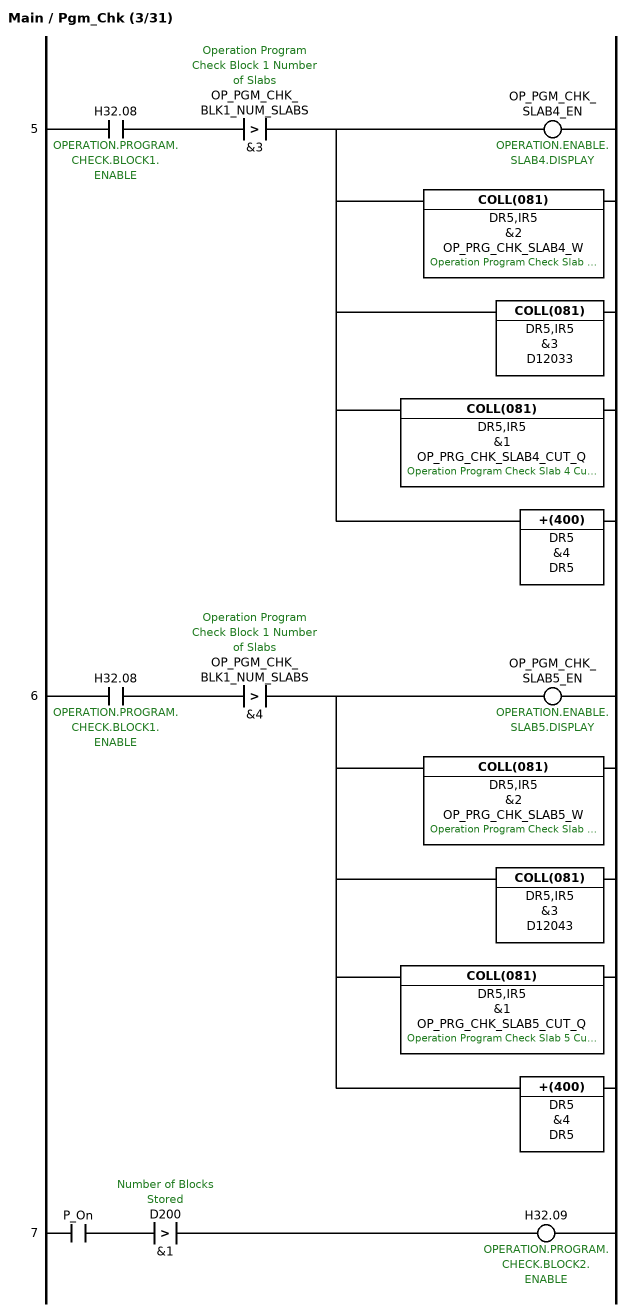
; [picture p96: Main / Pgm_Chk, rungs 5-7]
; rung 5
LD H32.08  ; OPERATION.PROGRAM.CHECK.BLOCK1.ENABLE
AND>(320) OP_PGM_CHK_BLK1_NUM_SLABS &3  ; Operation Program Check Block 1 Number of Slabs
OUT OP_PGM_CHK_SLAB4_EN  ; OPERATION.ENABLE.SLAB4.DISPLAY
COLL(081) DR5,IR5 &2 OP_PRG_CHK_SLAB4_W  ; Operation Program Check Slab 4 Width
COLL(081) DR5,IR5 &3 D12033
COLL(081) DR5,IR5 &1 OP_PRG_CHK_SLAB4_CUT_Q  ; Operation Program Check Slab 4 Cut Quantity
+(400) DR5 &4 DR5
; rung 6
LD H32.08  ; OPERATION.PROGRAM.CHECK.BLOCK1.ENABLE
AND>(320) OP_PGM_CHK_BLK1_NUM_SLABS &4  ; Operation Program Check Block 1 Number of Slabs
OUT OP_PGM_CHK_SLAB5_EN  ; OPERATION.ENABLE.SLAB5.DISPLAY
COLL(081) DR5,IR5 &2 OP_PRG_CHK_SLAB5_W  ; Operation Program Check Slab 5 Width
COLL(081) DR5,IR5 &3 D12043
COLL(081) DR5,IR5 &1 OP_PRG_CHK_SLAB5_CUT_Q  ; Operation Program Check Slab 5 Cut Quantity
+(400) DR5 &4 DR5
; rung 7
LD P_On
AND>(320) D200 &1  ; Number of Blocks Stored
OUT H32.09  ; OPERATION.PROGRAM.CHECK.BLOCK2.ENABLE

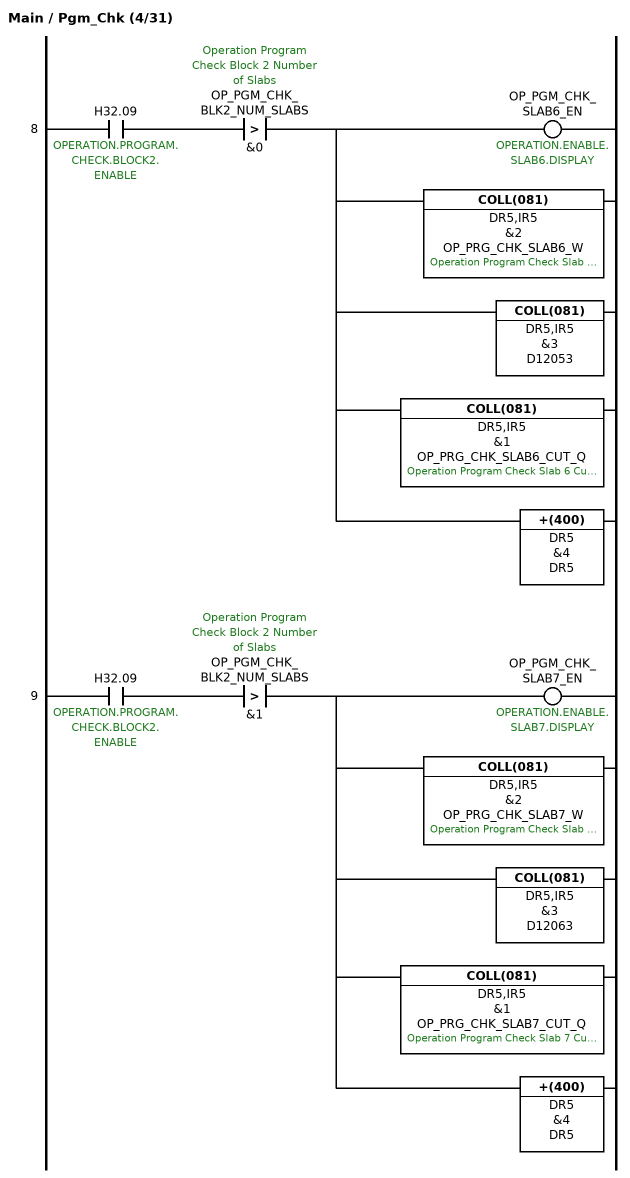
; rung 8
LD H32.09  ; OPERATION.PROGRAM.CHECK.BLOCK2.ENABLE
AND>(320) OP_PGM_CHK_BLK2_NUM_SLABS &0  ; Operation Program Check Block 2 Number of Slabs
OUT OP_PGM_CHK_SLAB6_EN  ; OPERATION.ENABLE.SLAB6.DISPLAY
COLL(081) DR5,IR5 &2 OP_PRG_CHK_SLAB6_W  ; Operation Program Check Slab 6 Width
COLL(081) DR5,IR5 &3 D12053
COLL(081) DR5,IR5 &1 OP_PRG_CHK_SLAB6_CUT_Q  ; Operation Program Check Slab 6 Cut Quantity
+(400) DR5 &4 DR5
; rung 9
LD H32.09  ; OPERATION.PROGRAM.CHECK.BLOCK2.ENABLE
AND>(320) OP_PGM_CHK_BLK2_NUM_SLABS &1  ; Operation Program Check Block 2 Number of Slabs
OUT OP_PGM_CHK_SLAB7_EN  ; OPERATION.ENABLE.SLAB7.DISPLAY
COLL(081) DR5,IR5 &2 OP_PRG_CHK_SLAB7_W  ; Operation Program Check Slab 7 Width
COLL(081) DR5,IR5 &3 D12063
COLL(081) DR5,IR5 &1 OP_PRG_CHK_SLAB7_CUT_Q  ; Operation Program Check Slab 7 Cut Quantity
+(400) DR5 &4 DR5

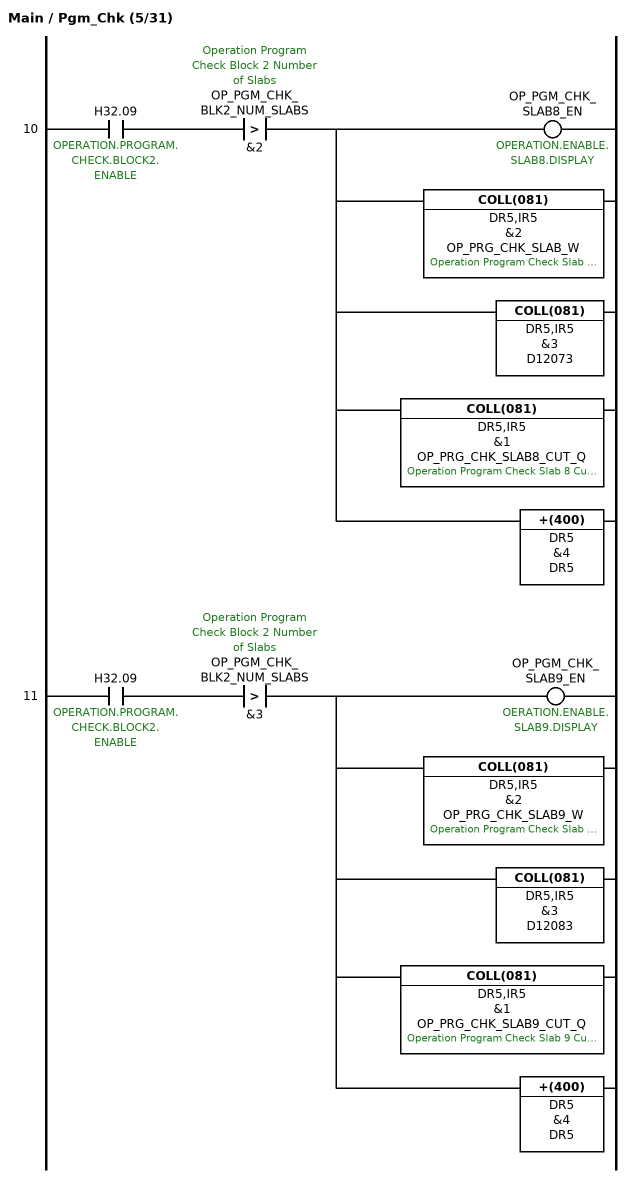
; rung 10
LD H32.09  ; OPERATION.PROGRAM.CHECK.BLOCK2.ENABLE
AND>(320) OP_PGM_CHK_BLK2_NUM_SLABS &2  ; Operation Program Check Block 2 Number of Slabs
OUT OP_PGM_CHK_SLAB8_EN  ; OPERATION.ENABLE.SLAB8.DISPLAY
COLL(081) DR5,IR5 &2 OP_PRG_CHK_SLAB_W  ; Operation Program Check Slab 8 Width
COLL(081) DR5,IR5 &3 D12073
COLL(081) DR5,IR5 &1 OP_PRG_CHK_SLAB8_CUT_Q  ; Operation Program Check Slab 8 Cut Quantity
+(400) DR5 &4 DR5
; rung 11
LD H32.09  ; OPERATION.PROGRAM.CHECK.BLOCK2.ENABLE
AND>(320) OP_PGM_CHK_BLK2_NUM_SLABS &3  ; Operation Program Check Block 2 Number of Slabs
OUT OP_PGM_CHK_SLAB9_EN  ; OERATION.ENABLE.SLAB9.DISPLAY
COLL(081) DR5,IR5 &2 OP_PRG_CHK_SLAB9_W  ; Operation Program Check Slab 9 Width
COLL(081) DR5,IR5 &3 D12083
COLL(081) DR5,IR5 &1 OP_PRG_CHK_SLAB9_CUT_Q  ; Operation Program Check Slab 9 Cut Quantity
+(400) DR5 &4 DR5

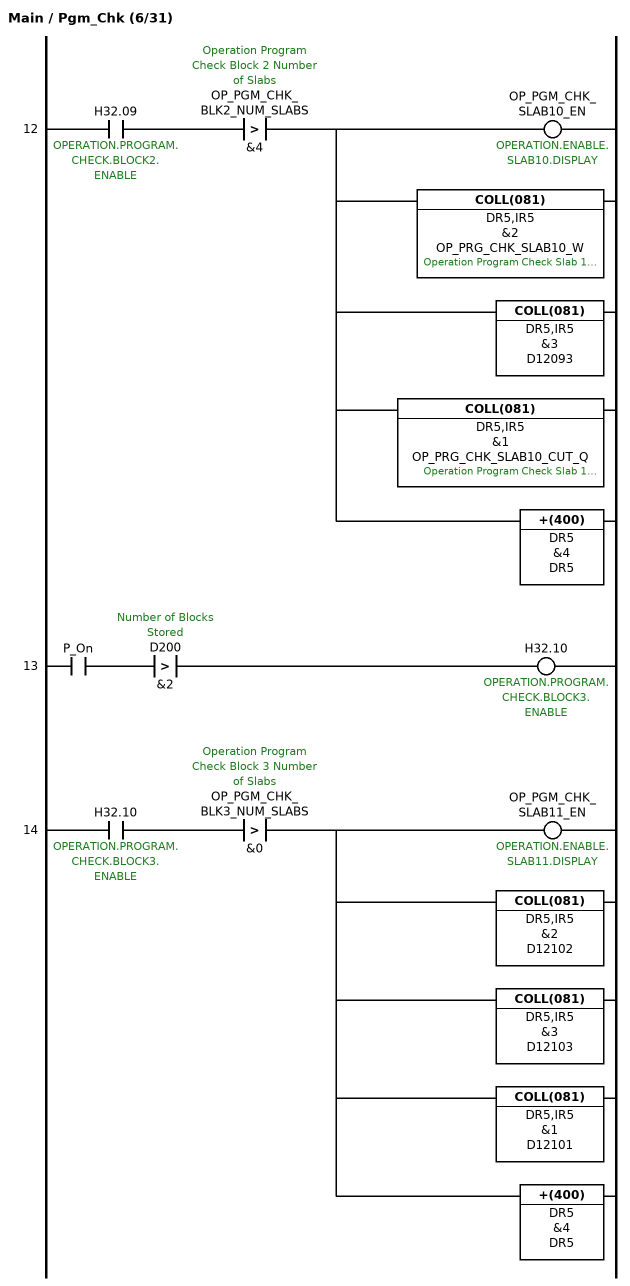
; rung 12
LD H32.09  ; OPERATION.PROGRAM.CHECK.BLOCK2.ENABLE
AND>(320) OP_PGM_CHK_BLK2_NUM_SLABS &4  ; Operation Program Check Block 2 Number of Slabs
OUT OP_PGM_CHK_SLAB10_EN  ; OPERATION.ENABLE.SLAB10.DISPLAY
COLL(081) DR5,IR5 &2 OP_PRG_CHK_SLAB10_W  ; Operation Program Check Slab 10 Width
COLL(081) DR5,IR5 &3 D12093
COLL(081) DR5,IR5 &1 OP_PRG_CHK_SLAB10_CUT_Q  ; Operation Program Check Slab 10 Cut Quantity
+(400) DR5 &4 DR5
; rung 13
LD P_On
AND>(320) D200 &2  ; Number of Blocks Stored
OUT H32.10  ; OPERATION.PROGRAM.CHECK.BLOCK3.ENABLE
; rung 14
LD H32.10  ; OPERATION.PROGRAM.CHECK.BLOCK3.ENABLE
AND>(320) OP_PGM_CHK_BLK3_NUM_SLABS &0  ; Operation Program Check Block 3 Number of Slabs
OUT OP_PGM_CHK_SLAB11_EN  ; OPERATION.ENABLE.SLAB11.DISPLAY
COLL(081) DR5,IR5 &2 D12102
COLL(081) DR5,IR5 &3 D12103
COLL(081) DR5,IR5 &1 D12101
+(400) DR5 &4 DR5

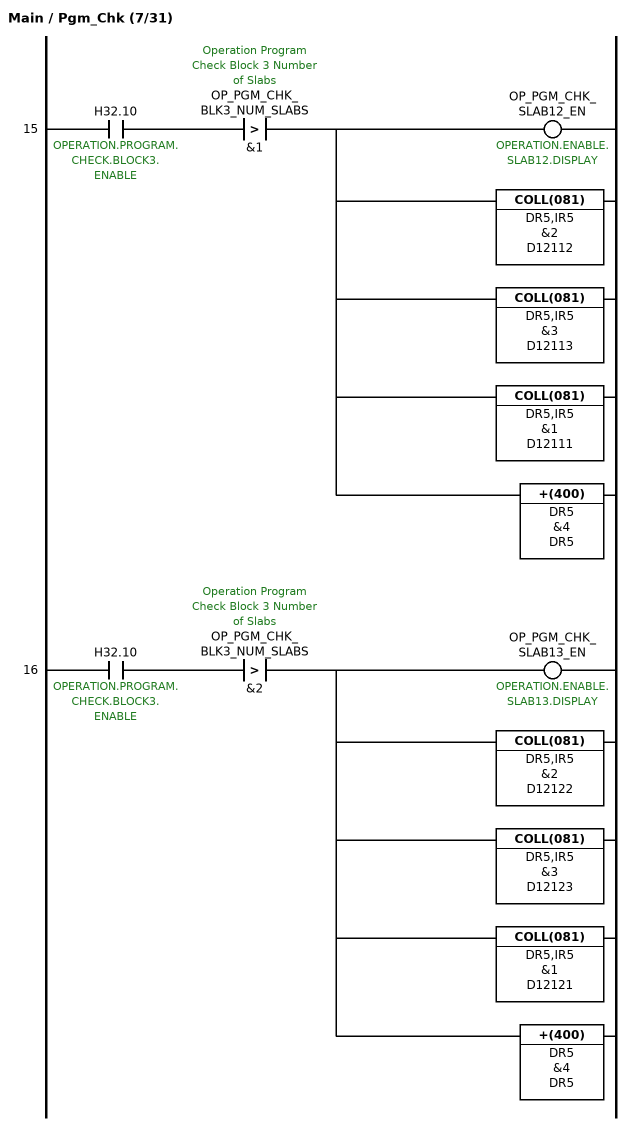
; rung 15
LD H32.10  ; OPERATION.PROGRAM.CHECK.BLOCK3.ENABLE
AND>(320) OP_PGM_CHK_BLK3_NUM_SLABS &1  ; Operation Program Check Block 3 Number of Slabs
OUT OP_PGM_CHK_SLAB12_EN  ; OPERATION.ENABLE.SLAB12.DISPLAY
COLL(081) DR5,IR5 &2 D12112
COLL(081) DR5,IR5 &3 D12113
COLL(081) DR5,IR5 &1 D12111
+(400) DR5 &4 DR5
; rung 16
LD H32.10  ; OPERATION.PROGRAM.CHECK.BLOCK3.ENABLE
AND>(320) OP_PGM_CHK_BLK3_NUM_SLABS &2  ; Operation Program Check Block 3 Number of Slabs
OUT OP_PGM_CHK_SLAB13_EN  ; OPERATION.ENABLE.SLAB13.DISPLAY
COLL(081) DR5,IR5 &2 D12122
COLL(081) DR5,IR5 &3 D12123
COLL(081) DR5,IR5 &1 D12121
+(400) DR5 &4 DR5

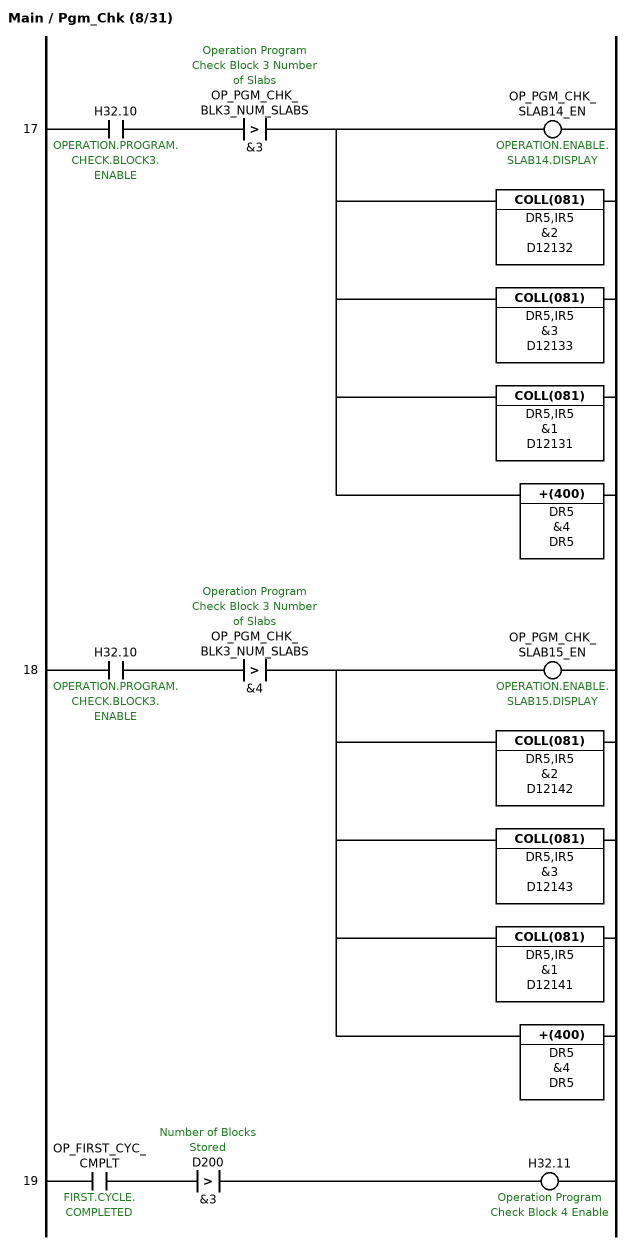
; rung 17
LD H32.10  ; OPERATION.PROGRAM.CHECK.BLOCK3.ENABLE
AND>(320) OP_PGM_CHK_BLK3_NUM_SLABS &3  ; Operation Program Check Block 3 Number of Slabs
OUT OP_PGM_CHK_SLAB14_EN  ; OPERATION.ENABLE.SLAB14.DISPLAY
COLL(081) DR5,IR5 &2 D12132
COLL(081) DR5,IR5 &3 D12133
COLL(081) DR5,IR5 &1 D12131
+(400) DR5 &4 DR5
; rung 18
LD H32.10  ; OPERATION.PROGRAM.CHECK.BLOCK3.ENABLE
AND>(320) OP_PGM_CHK_BLK3_NUM_SLABS &4  ; Operation Program Check Block 3 Number of Slabs
OUT OP_PGM_CHK_SLAB15_EN  ; OPERATION.ENABLE.SLAB15.DISPLAY
COLL(081) DR5,IR5 &2 D12142
COLL(081) DR5,IR5 &3 D12143
COLL(081) DR5,IR5 &1 D12141
+(400) DR5 &4 DR5
; rung 19
LD OP_FIRST_CYC_CMPLT  ; FIRST.CYCLE.COMPLETED
AND>(320) D200 &3  ; Number of Blocks Stored
OUT H32.11  ; Operation Program Check Block 4 Enable

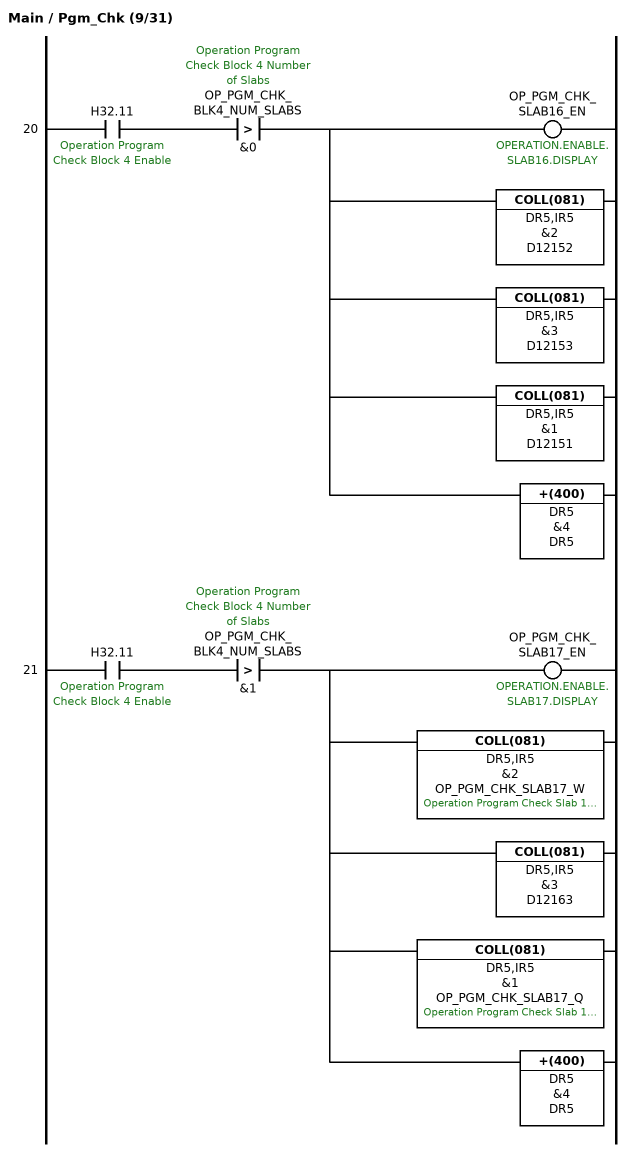
; rung 20
LD H32.11  ; Operation Program Check Block 4 Enable
AND>(320) OP_PGM_CHK_BLK4_NUM_SLABS &0  ; Operation Program Check Block 4 Number of Slabs
OUT OP_PGM_CHK_SLAB16_EN  ; OPERATION.ENABLE.SLAB16.DISPLAY
COLL(081) DR5,IR5 &2 D12152
COLL(081) DR5,IR5 &3 D12153
COLL(081) DR5,IR5 &1 D12151
+(400) DR5 &4 DR5
; rung 21
LD H32.11  ; Operation Program Check Block 4 Enable
AND>(320) OP_PGM_CHK_BLK4_NUM_SLABS &1  ; Operation Program Check Block 4 Number of Slabs
OUT OP_PGM_CHK_SLAB17_EN  ; OPERATION.ENABLE.SLAB17.DISPLAY
COLL(081) DR5,IR5 &2 OP_PGM_CHK_SLAB17_W  ; Operation Program Check Slab 17 Size
COLL(081) DR5,IR5 &3 D12163
COLL(081) DR5,IR5 &1 OP_PGM_CHK_SLAB17_Q  ; Operation Program Check Slab 17 Quantity
+(400) DR5 &4 DR5

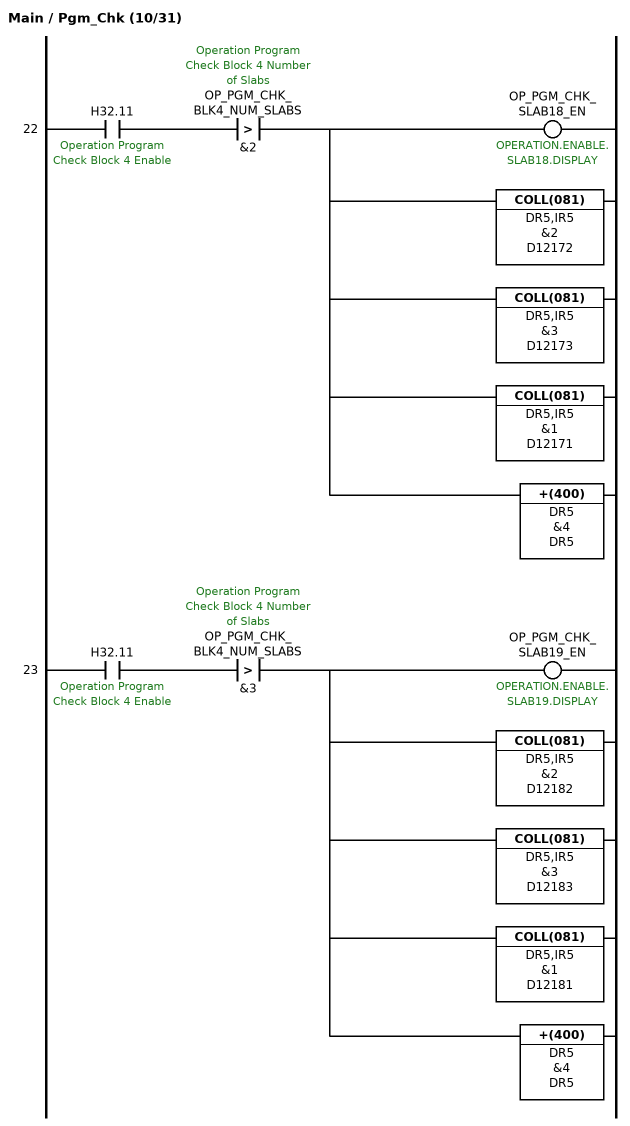
; rung 22
LD H32.11  ; Operation Program Check Block 4 Enable
AND>(320) OP_PGM_CHK_BLK4_NUM_SLABS &2  ; Operation Program Check Block 4 Number of Slabs
OUT OP_PGM_CHK_SLAB18_EN  ; OPERATION.ENABLE.SLAB18.DISPLAY
COLL(081) DR5,IR5 &2 D12172
COLL(081) DR5,IR5 &3 D12173
COLL(081) DR5,IR5 &1 D12171
+(400) DR5 &4 DR5
; rung 23
LD H32.11  ; Operation Program Check Block 4 Enable
AND>(320) OP_PGM_CHK_BLK4_NUM_SLABS &3  ; Operation Program Check Block 4 Number of Slabs
OUT OP_PGM_CHK_SLAB19_EN  ; OPERATION.ENABLE.SLAB19.DISPLAY
COLL(081) DR5,IR5 &2 D12182
COLL(081) DR5,IR5 &3 D12183
COLL(081) DR5,IR5 &1 D12181
+(400) DR5 &4 DR5

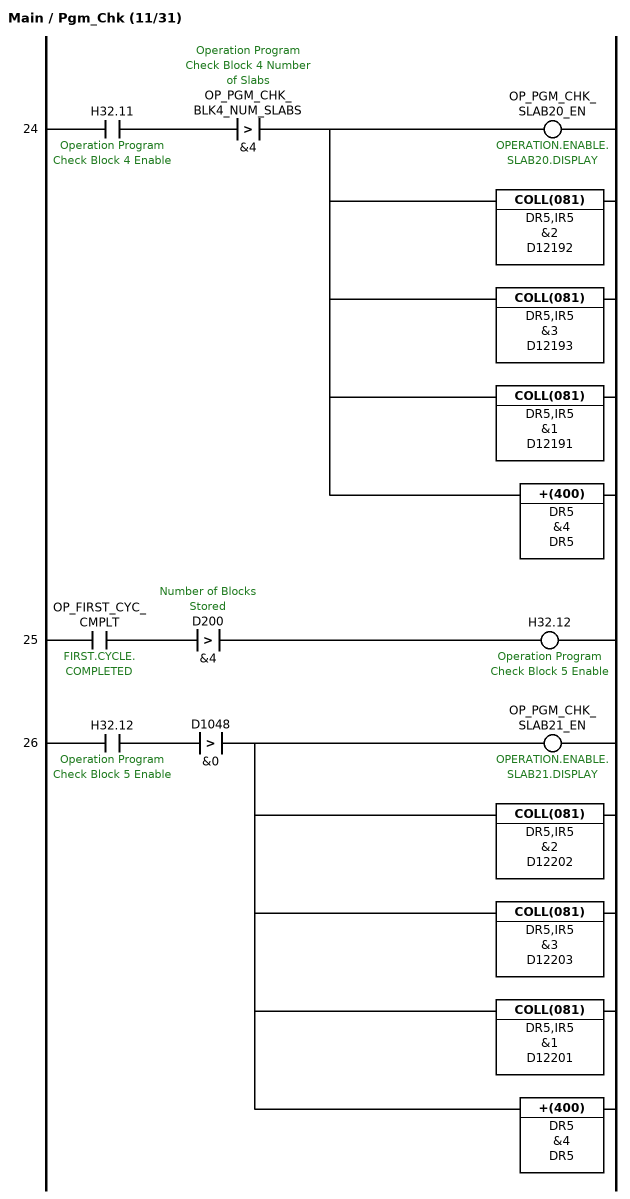
; rung 24
LD H32.11  ; Operation Program Check Block 4 Enable
AND>(320) OP_PGM_CHK_BLK4_NUM_SLABS &4  ; Operation Program Check Block 4 Number of Slabs
OUT OP_PGM_CHK_SLAB20_EN  ; OPERATION.ENABLE.SLAB20.DISPLAY
COLL(081) DR5,IR5 &2 D12192
COLL(081) DR5,IR5 &3 D12193
COLL(081) DR5,IR5 &1 D12191
+(400) DR5 &4 DR5
; rung 25
LD OP_FIRST_CYC_CMPLT  ; FIRST.CYCLE.COMPLETED
AND>(320) D200 &4  ; Number of Blocks Stored
OUT H32.12  ; Operation Program Check Block 5 Enable
; rung 26
LD H32.12  ; Operation Program Check Block 5 Enable
AND>(320) D1048 &0
OUT OP_PGM_CHK_SLAB21_EN  ; OPERATION.ENABLE.SLAB21.DISPLAY
COLL(081) DR5,IR5 &2 D12202
COLL(081) DR5,IR5 &3 D12203
COLL(081) DR5,IR5 &1 D12201
+(400) DR5 &4 DR5

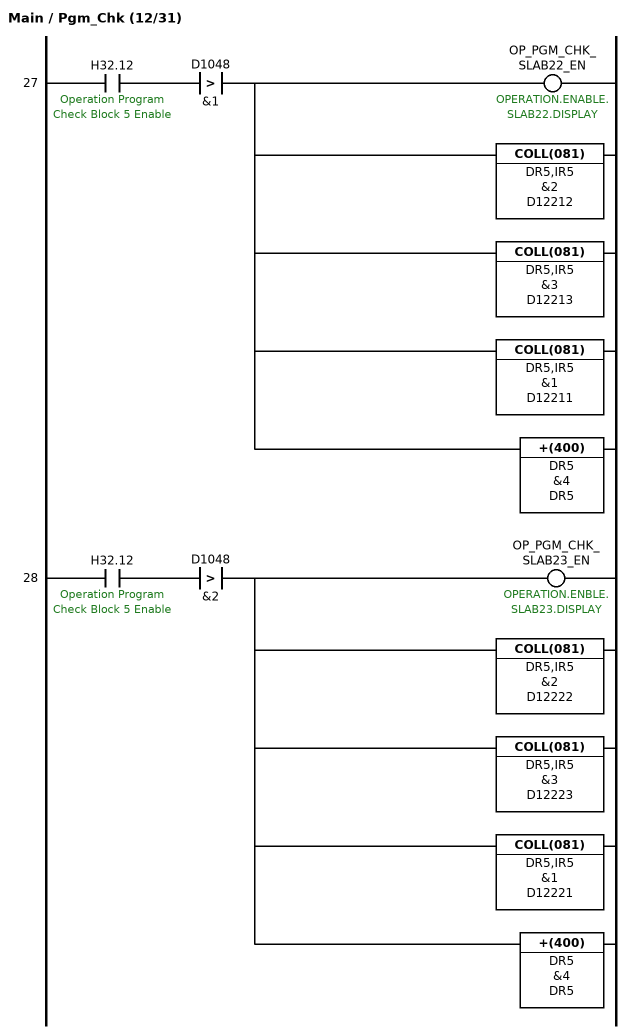
; rung 27
LD H32.12  ; Operation Program Check Block 5 Enable
AND>(320) D1048 &1
OUT OP_PGM_CHK_SLAB22_EN  ; OPERATION.ENABLE.SLAB22.DISPLAY
COLL(081) DR5,IR5 &2 D12212
COLL(081) DR5,IR5 &3 D12213
COLL(081) DR5,IR5 &1 D12211
+(400) DR5 &4 DR5
; rung 28
LD H32.12  ; Operation Program Check Block 5 Enable
AND>(320) D1048 &2
OUT OP_PGM_CHK_SLAB23_EN  ; OPERATION.ENBLE.SLAB23.DISPLAY
COLL(081) DR5,IR5 &2 D12222
COLL(081) DR5,IR5 &3 D12223
COLL(081) DR5,IR5 &1 D12221
+(400) DR5 &4 DR5

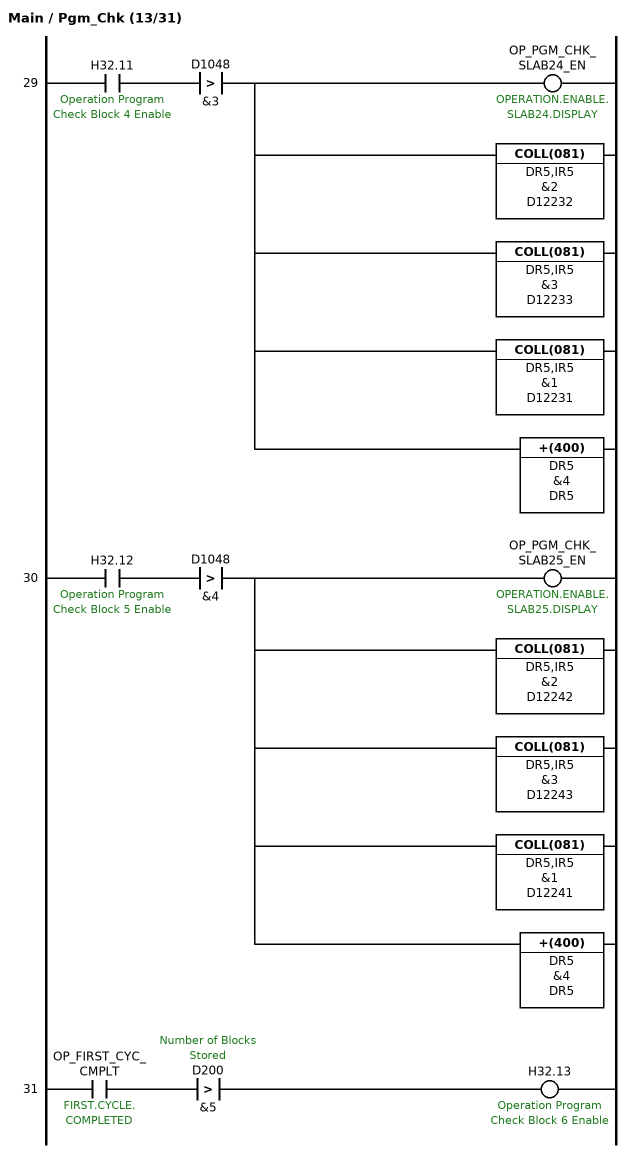
; rung 29
LD H32.11  ; Operation Program Check Block 4 Enable
AND>(320) D1048 &3
OUT OP_PGM_CHK_SLAB24_EN  ; OPERATION.ENABLE.SLAB24.DISPLAY
COLL(081) DR5,IR5 &2 D12232
COLL(081) DR5,IR5 &3 D12233
COLL(081) DR5,IR5 &1 D12231
+(400) DR5 &4 DR5
; rung 30
LD H32.12  ; Operation Program Check Block 5 Enable
AND>(320) D1048 &4
OUT OP_PGM_CHK_SLAB25_EN  ; OPERATION.ENABLE.SLAB25.DISPLAY
COLL(081) DR5,IR5 &2 D12242
COLL(081) DR5,IR5 &3 D12243
COLL(081) DR5,IR5 &1 D12241
+(400) DR5 &4 DR5
; rung 31
LD OP_FIRST_CYC_CMPLT  ; FIRST.CYCLE.COMPLETED
AND>(320) D200 &5  ; Number of Blocks Stored
OUT H32.13  ; Operation Program Check Block 6 Enable

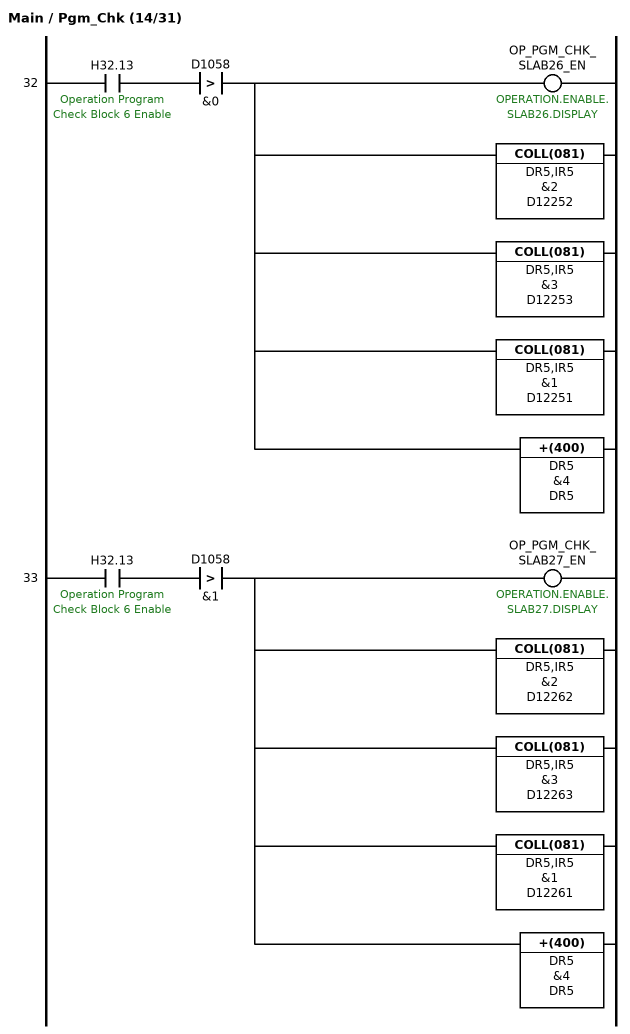
; rung 32
LD H32.13  ; Operation Program Check Block 6 Enable
AND>(320) D1058 &0
OUT OP_PGM_CHK_SLAB26_EN  ; OPERATION.ENABLE.SLAB26.DISPLAY
COLL(081) DR5,IR5 &2 D12252
COLL(081) DR5,IR5 &3 D12253
COLL(081) DR5,IR5 &1 D12251
+(400) DR5 &4 DR5
; rung 33
LD H32.13  ; Operation Program Check Block 6 Enable
AND>(320) D1058 &1
OUT OP_PGM_CHK_SLAB27_EN  ; OPERATION.ENABLE.SLAB27.DISPLAY
COLL(081) DR5,IR5 &2 D12262
COLL(081) DR5,IR5 &3 D12263
COLL(081) DR5,IR5 &1 D12261
+(400) DR5 &4 DR5

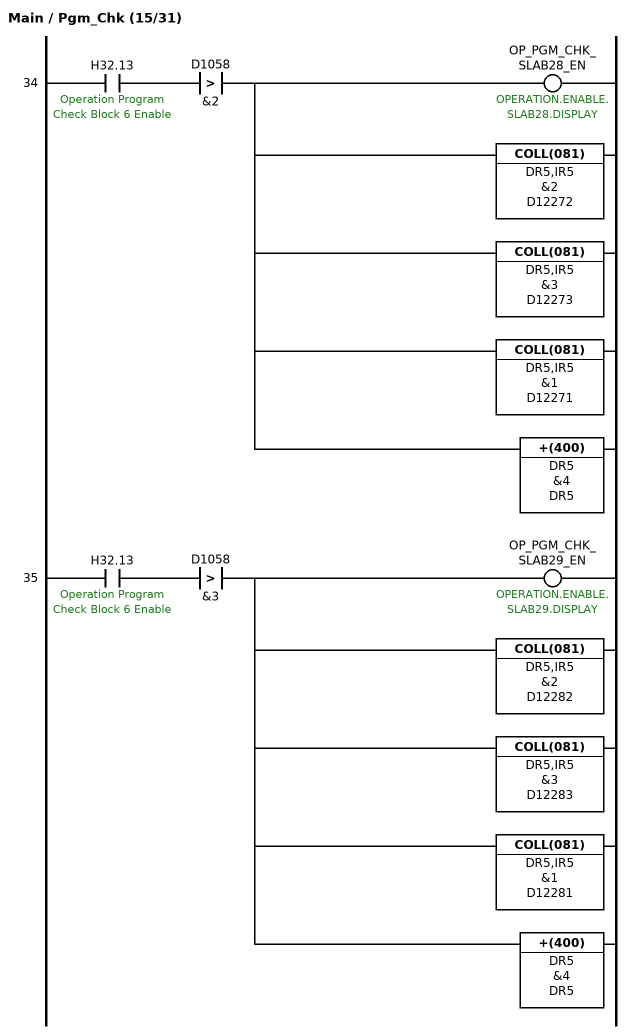
; rung 34
LD H32.13  ; Operation Program Check Block 6 Enable
AND>(320) D1058 &2
OUT OP_PGM_CHK_SLAB28_EN  ; OPERATION.ENABLE.SLAB28.DISPLAY
COLL(081) DR5,IR5 &2 D12272
COLL(081) DR5,IR5 &3 D12273
COLL(081) DR5,IR5 &1 D12271
+(400) DR5 &4 DR5
; rung 35
LD H32.13  ; Operation Program Check Block 6 Enable
AND>(320) D1058 &3
OUT OP_PGM_CHK_SLAB29_EN  ; OPERATION.ENABLE.SLAB29.DISPLAY
COLL(081) DR5,IR5 &2 D12282
COLL(081) DR5,IR5 &3 D12283
COLL(081) DR5,IR5 &1 D12281
+(400) DR5 &4 DR5

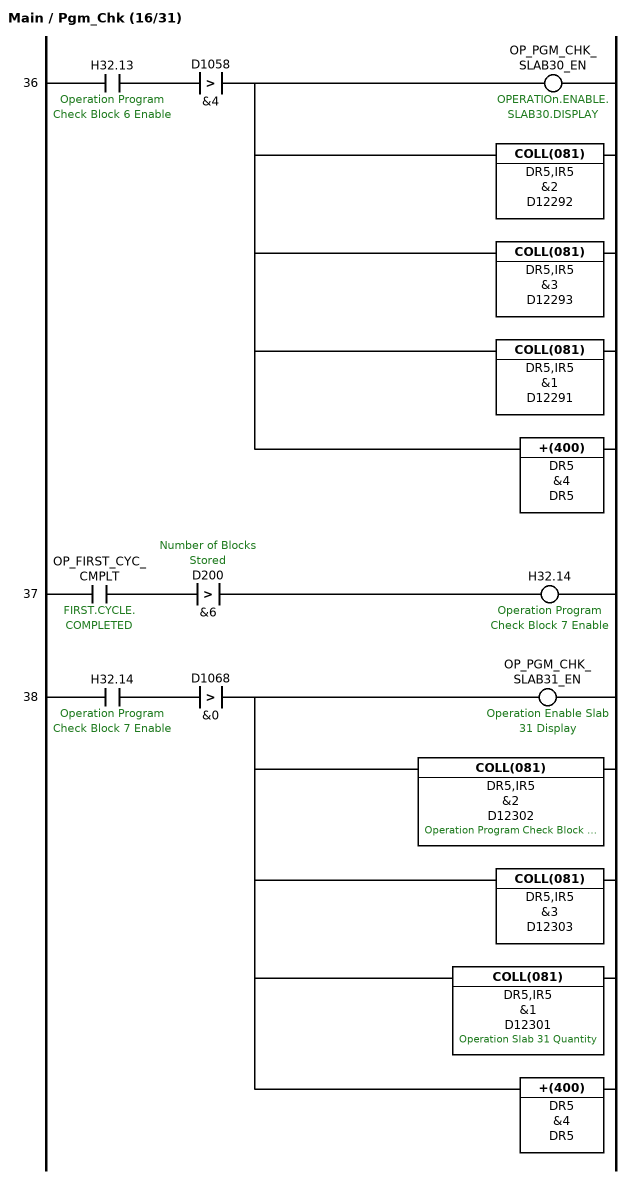
; rung 36
LD H32.13  ; Operation Program Check Block 6 Enable
AND>(320) D1058 &4
OUT OP_PGM_CHK_SLAB30_EN  ; OPERATIOn.ENABLE.SLAB30.DISPLAY
COLL(081) DR5,IR5 &2 D12292
COLL(081) DR5,IR5 &3 D12293
COLL(081) DR5,IR5 &1 D12291
+(400) DR5 &4 DR5
; rung 37
LD OP_FIRST_CYC_CMPLT  ; FIRST.CYCLE.COMPLETED
AND>(320) D200 &6  ; Number of Blocks Stored
OUT H32.14  ; Operation Program Check Block 7 Enable
; rung 38
LD H32.14  ; Operation Program Check Block 7 Enable
AND>(320) D1068 &0
OUT OP_PGM_CHK_SLAB31_EN  ; Operation Enable Slab 31 Display
COLL(081) DR5,IR5 &2 D12302  ; Operation Program Check Block 7 Slab 31 Width
COLL(081) DR5,IR5 &3 D12303
COLL(081) DR5,IR5 &1 D12301  ; Operation Slab 31 Quantity
+(400) DR5 &4 DR5

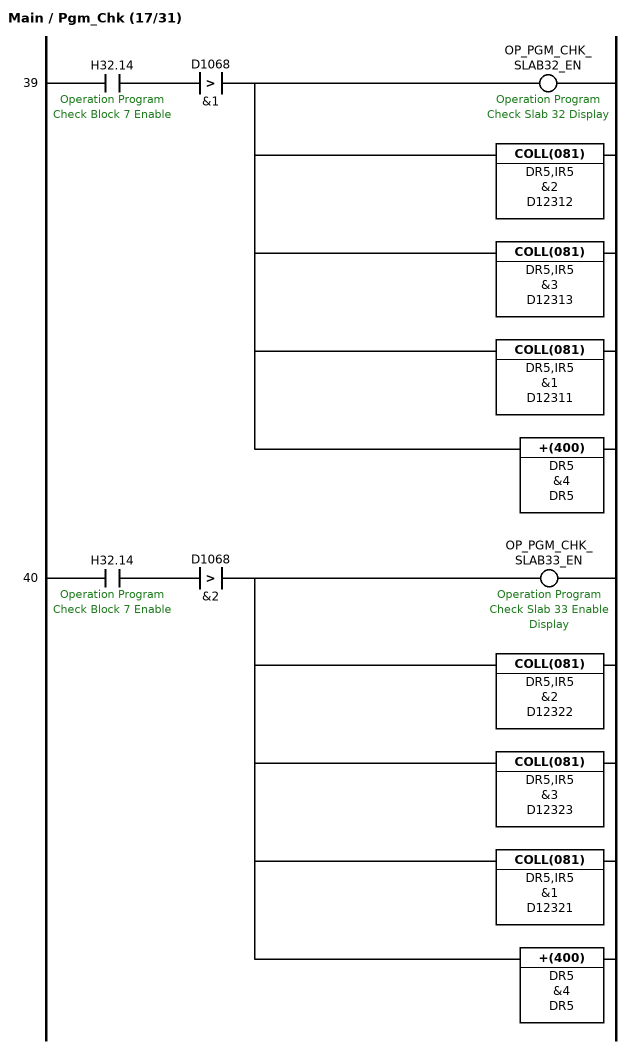
; rung 39
LD H32.14  ; Operation Program Check Block 7 Enable
AND>(320) D1068 &1
OUT OP_PGM_CHK_SLAB32_EN  ; Operation Program Check Slab 32 Display
COLL(081) DR5,IR5 &2 D12312
COLL(081) DR5,IR5 &3 D12313
COLL(081) DR5,IR5 &1 D12311
+(400) DR5 &4 DR5
; rung 40
LD H32.14  ; Operation Program Check Block 7 Enable
AND>(320) D1068 &2
OUT OP_PGM_CHK_SLAB33_EN  ; Operation Program Check Slab 33 Enable Display
COLL(081) DR5,IR5 &2 D12322
COLL(081) DR5,IR5 &3 D12323
COLL(081) DR5,IR5 &1 D12321
+(400) DR5 &4 DR5

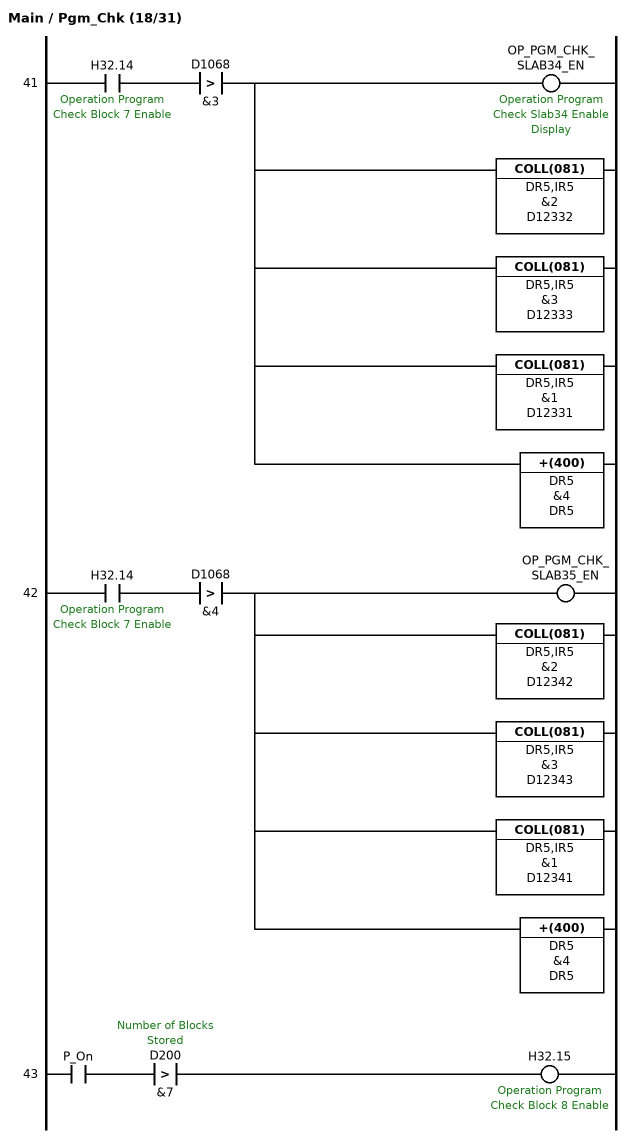
; rung 41
LD H32.14  ; Operation Program Check Block 7 Enable
AND>(320) D1068 &3
OUT OP_PGM_CHK_SLAB34_EN  ; Operation Program Check Slab34 Enable Display
COLL(081) DR5,IR5 &2 D12332
COLL(081) DR5,IR5 &3 D12333
COLL(081) DR5,IR5 &1 D12331
+(400) DR5 &4 DR5
; rung 42
LD H32.14  ; Operation Program Check Block 7 Enable
AND>(320) D1068 &4
OUT OP_PGM_CHK_SLAB35_EN
COLL(081) DR5,IR5 &2 D12342
COLL(081) DR5,IR5 &3 D12343
COLL(081) DR5,IR5 &1 D12341
+(400) DR5 &4 DR5
; rung 43
LD P_On
AND>(320) D200 &7  ; Number of Blocks Stored
OUT H32.15  ; Operation Program Check Block 8 Enable

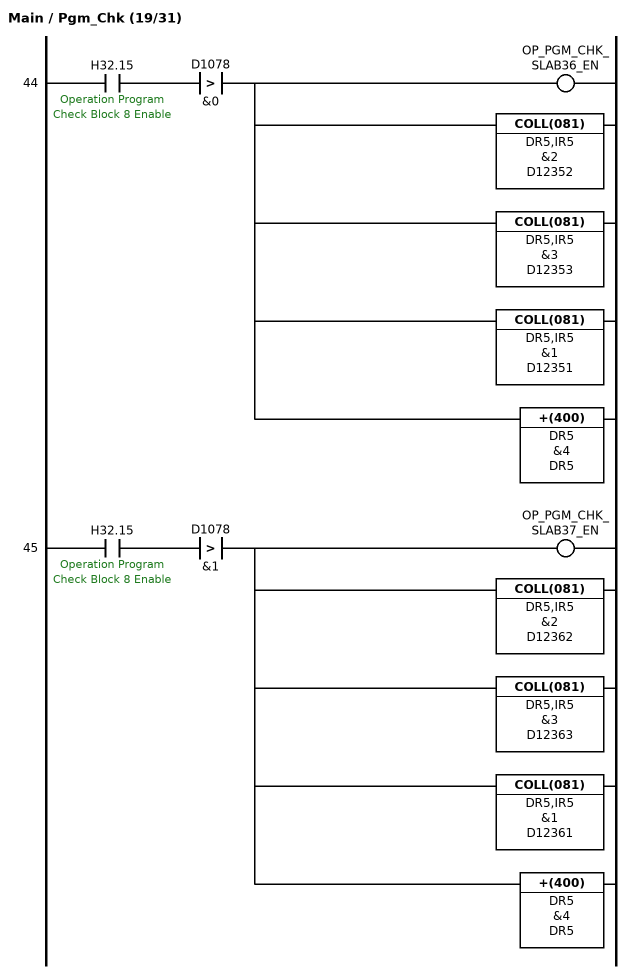
; rung 44
LD H32.15  ; Operation Program Check Block 8 Enable
AND>(320) D1078 &0
OUT OP_PGM_CHK_SLAB36_EN
COLL(081) DR5,IR5 &2 D12352
COLL(081) DR5,IR5 &3 D12353
COLL(081) DR5,IR5 &1 D12351
+(400) DR5 &4 DR5
; rung 45
LD H32.15  ; Operation Program Check Block 8 Enable
AND>(320) D1078 &1
OUT OP_PGM_CHK_SLAB37_EN
COLL(081) DR5,IR5 &2 D12362
COLL(081) DR5,IR5 &3 D12363
COLL(081) DR5,IR5 &1 D12361
+(400) DR5 &4 DR5

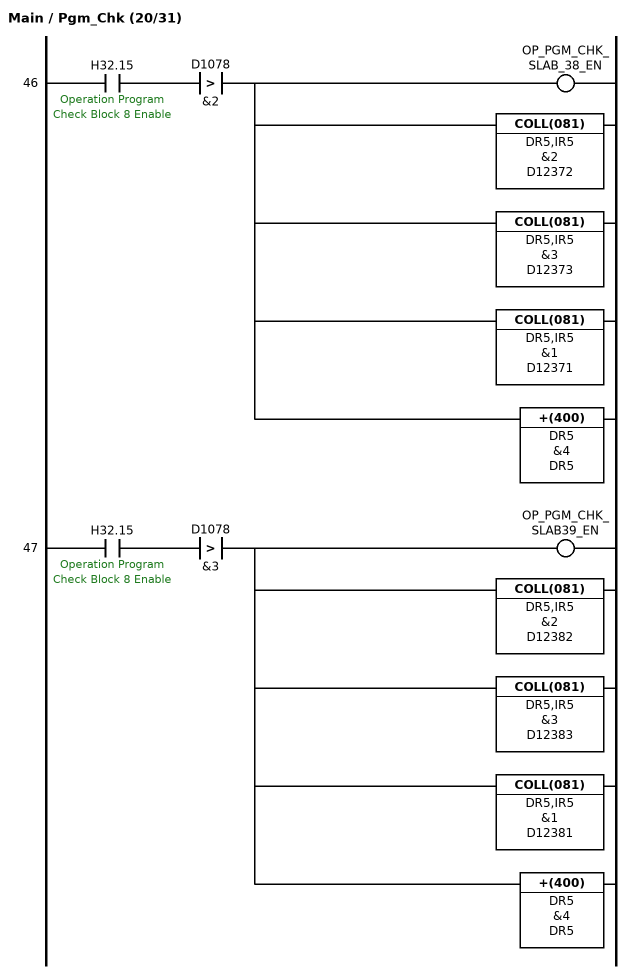
; rung 46
LD H32.15  ; Operation Program Check Block 8 Enable
AND>(320) D1078 &2
OUT OP_PGM_CHK_SLAB_38_EN
COLL(081) DR5,IR5 &2 D12372
COLL(081) DR5,IR5 &3 D12373
COLL(081) DR5,IR5 &1 D12371
+(400) DR5 &4 DR5
; rung 47
LD H32.15  ; Operation Program Check Block 8 Enable
AND>(320) D1078 &3
OUT OP_PGM_CHK_SLAB39_EN
COLL(081) DR5,IR5 &2 D12382
COLL(081) DR5,IR5 &3 D12383
COLL(081) DR5,IR5 &1 D12381
+(400) DR5 &4 DR5

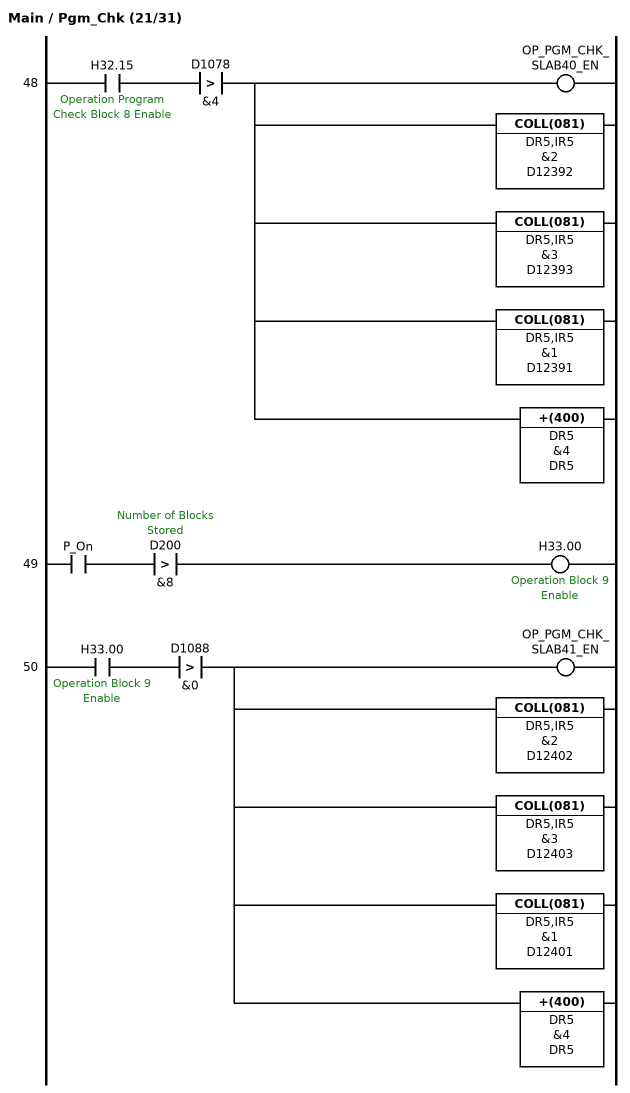
; rung 48
LD H32.15  ; Operation Program Check Block 8 Enable
AND>(320) D1078 &4
OUT OP_PGM_CHK_SLAB40_EN
COLL(081) DR5,IR5 &2 D12392
COLL(081) DR5,IR5 &3 D12393
COLL(081) DR5,IR5 &1 D12391
+(400) DR5 &4 DR5
; rung 49
LD P_On
AND>(320) D200 &8  ; Number of Blocks Stored
OUT H33.00  ; Operation Block 9 Enable
; rung 50
LD H33.00  ; Operation Block 9 Enable
AND>(320) D1088 &0
OUT OP_PGM_CHK_SLAB41_EN
COLL(081) DR5,IR5 &2 D12402
COLL(081) DR5,IR5 &3 D12403
COLL(081) DR5,IR5 &1 D12401
+(400) DR5 &4 DR5

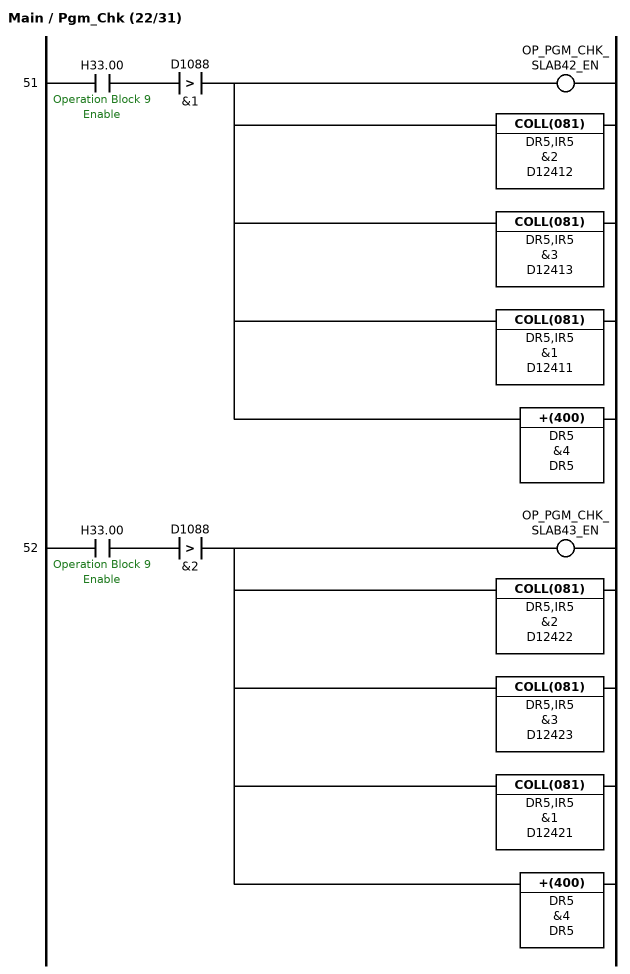
; rung 51
LD H33.00  ; Operation Block 9 Enable
AND>(320) D1088 &1
OUT OP_PGM_CHK_SLAB42_EN
COLL(081) DR5,IR5 &2 D12412
COLL(081) DR5,IR5 &3 D12413
COLL(081) DR5,IR5 &1 D12411
+(400) DR5 &4 DR5
; rung 52
LD H33.00  ; Operation Block 9 Enable
AND>(320) D1088 &2
OUT OP_PGM_CHK_SLAB43_EN
COLL(081) DR5,IR5 &2 D12422
COLL(081) DR5,IR5 &3 D12423
COLL(081) DR5,IR5 &1 D12421
+(400) DR5 &4 DR5

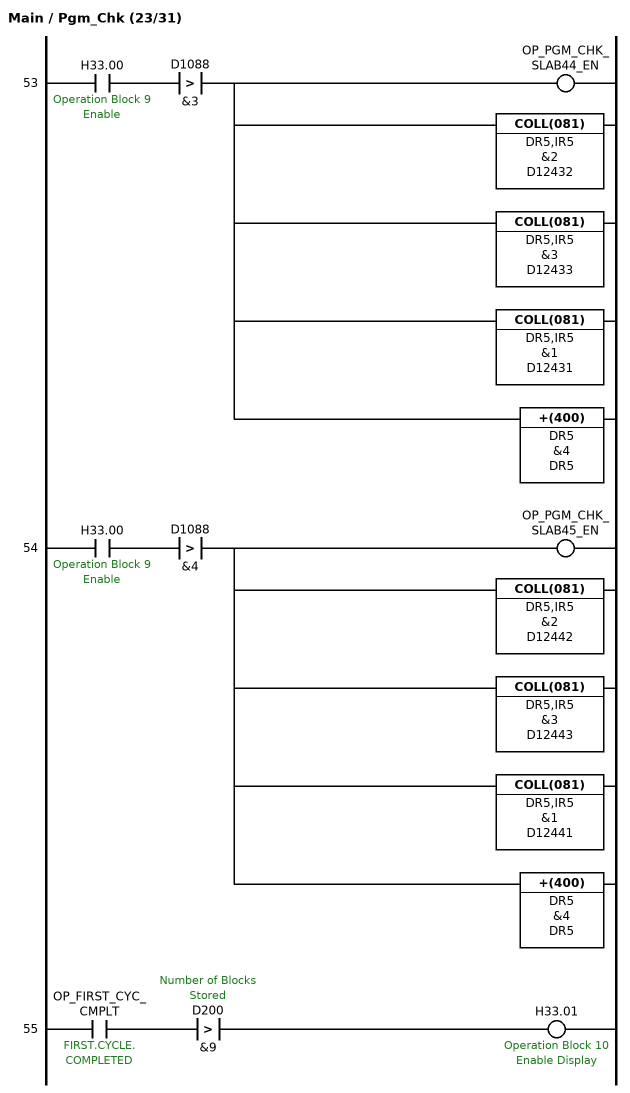
; rung 53
LD H33.00  ; Operation Block 9 Enable
AND>(320) D1088 &3
OUT OP_PGM_CHK_SLAB44_EN
COLL(081) DR5,IR5 &2 D12432
COLL(081) DR5,IR5 &3 D12433
COLL(081) DR5,IR5 &1 D12431
+(400) DR5 &4 DR5
; rung 54
LD H33.00  ; Operation Block 9 Enable
AND>(320) D1088 &4
OUT OP_PGM_CHK_SLAB45_EN
COLL(081) DR5,IR5 &2 D12442
COLL(081) DR5,IR5 &3 D12443
COLL(081) DR5,IR5 &1 D12441
+(400) DR5 &4 DR5
; rung 55
LD OP_FIRST_CYC_CMPLT  ; FIRST.CYCLE.COMPLETED
AND>(320) D200 &9  ; Number of Blocks Stored
OUT H33.01  ; Operation Block 10 Enable Display

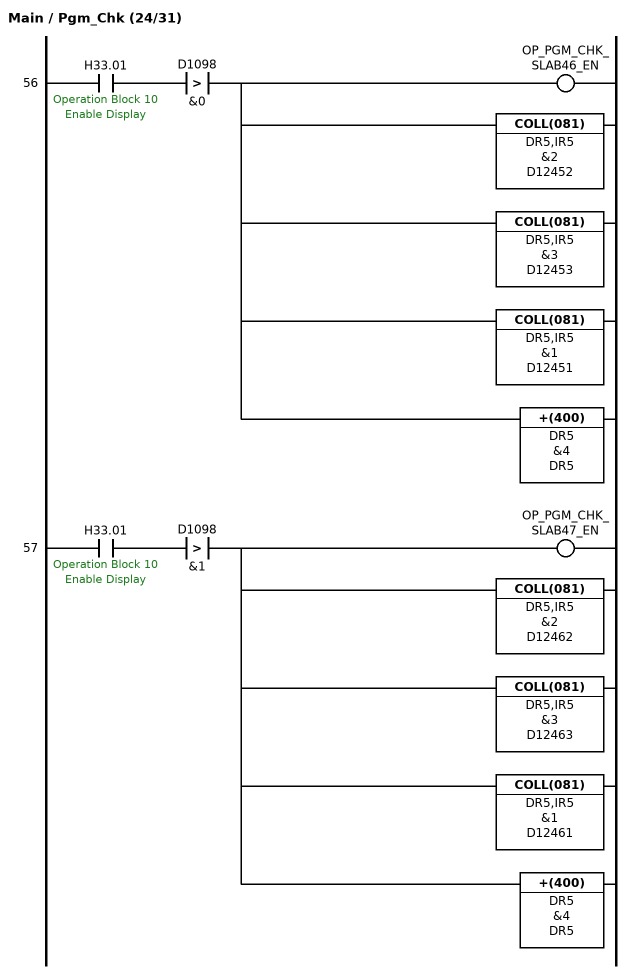
; rung 56
LD H33.01  ; Operation Block 10 Enable Display
AND>(320) D1098 &0
OUT OP_PGM_CHK_SLAB46_EN
COLL(081) DR5,IR5 &2 D12452
COLL(081) DR5,IR5 &3 D12453
COLL(081) DR5,IR5 &1 D12451
+(400) DR5 &4 DR5
; rung 57
LD H33.01  ; Operation Block 10 Enable Display
AND>(320) D1098 &1
OUT OP_PGM_CHK_SLAB47_EN
COLL(081) DR5,IR5 &2 D12462
COLL(081) DR5,IR5 &3 D12463
COLL(081) DR5,IR5 &1 D12461
+(400) DR5 &4 DR5

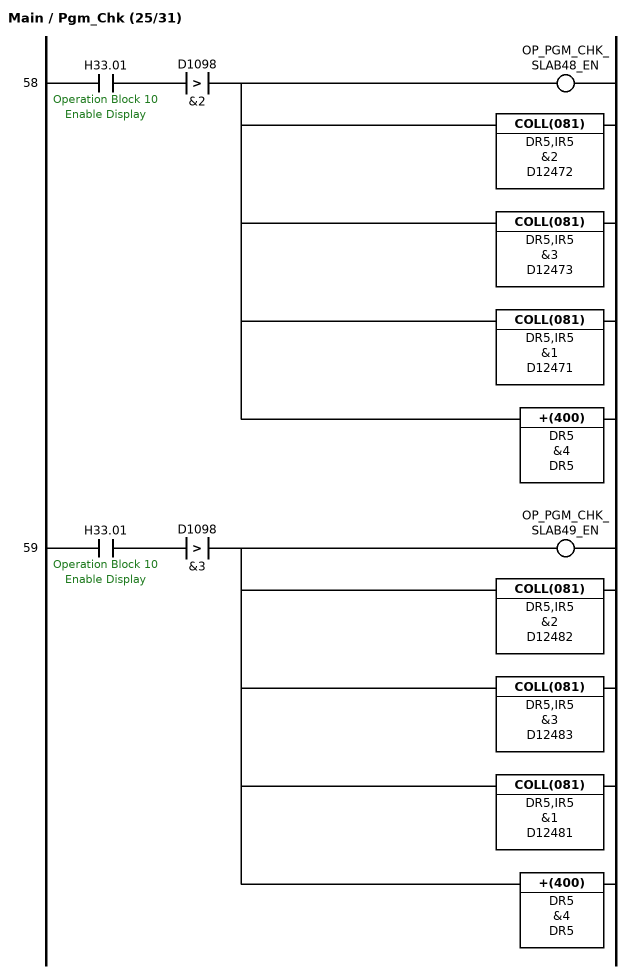
; rung 58
LD H33.01  ; Operation Block 10 Enable Display
AND>(320) D1098 &2
OUT OP_PGM_CHK_SLAB48_EN
COLL(081) DR5,IR5 &2 D12472
COLL(081) DR5,IR5 &3 D12473
COLL(081) DR5,IR5 &1 D12471
+(400) DR5 &4 DR5
; rung 59
LD H33.01  ; Operation Block 10 Enable Display
AND>(320) D1098 &3
OUT OP_PGM_CHK_SLAB49_EN
COLL(081) DR5,IR5 &2 D12482
COLL(081) DR5,IR5 &3 D12483
COLL(081) DR5,IR5 &1 D12481
+(400) DR5 &4 DR5

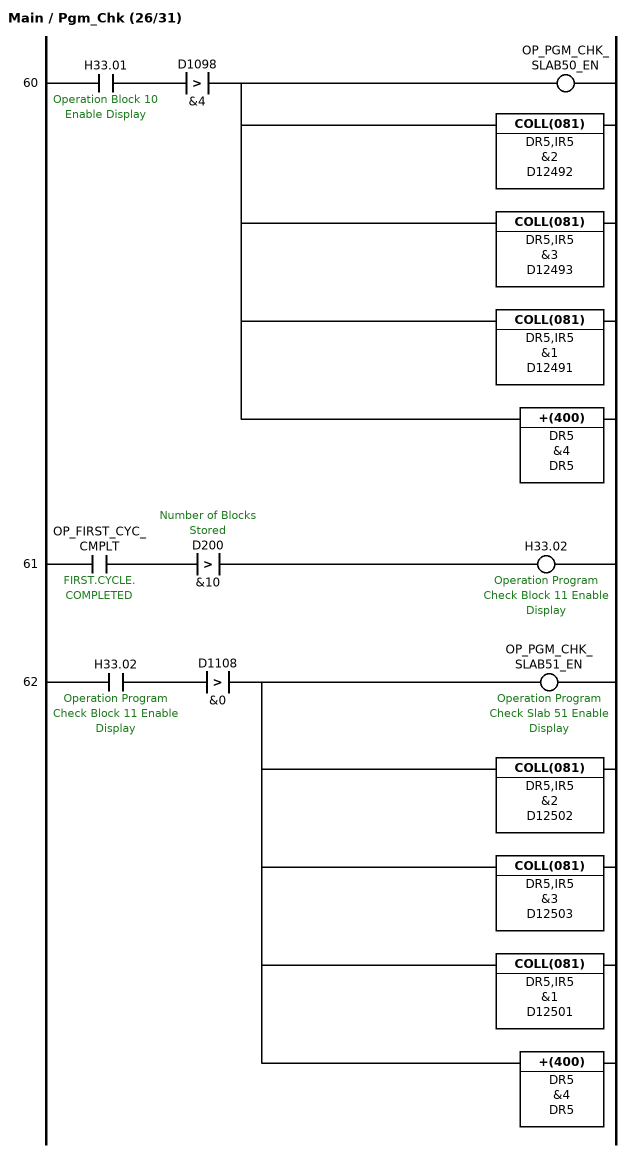
; rung 60
LD H33.01  ; Operation Block 10 Enable Display
AND>(320) D1098 &4
OUT OP_PGM_CHK_SLAB50_EN
COLL(081) DR5,IR5 &2 D12492
COLL(081) DR5,IR5 &3 D12493
COLL(081) DR5,IR5 &1 D12491
+(400) DR5 &4 DR5
; rung 61
LD OP_FIRST_CYC_CMPLT  ; FIRST.CYCLE.COMPLETED
AND>(320) D200 &10  ; Number of Blocks Stored
OUT H33.02  ; Operation Program Check Block 11 Enable Display
; rung 62
LD H33.02  ; Operation Program Check Block 11 Enable Display
AND>(320) D1108 &0
OUT OP_PGM_CHK_SLAB51_EN  ; Operation Program Check Slab 51 Enable Display
COLL(081) DR5,IR5 &2 D12502
COLL(081) DR5,IR5 &3 D12503
COLL(081) DR5,IR5 &1 D12501
+(400) DR5 &4 DR5

